FUNCTION_BLOCK ValveDynamics
VAR_INPUT
	udcv_IN : LREAL;
END_VAR
VAR_OUTPUT
	DynamicValve : LREAL;
END_VAR
VAR
	Timer : LREAL;
END_VAR

Timer := Timer + 0.001;

//Valve opening signal is sent through this
DynamicValve := ((100*SQRT(3))/SQRT(17))*EXP(-21*Timer)*SIN(3*SQRT(51)*Timer);

END_FUNCTION_BLOCK

(* stored: Version 1.1.0.1, ProductVersion 3.1.4024.9
   POU ValveDynamics: Id {bdd402cd-9955-422d-9429-c814b00ee090}, SpecialFunc None *)
